{attribute 'GeneratedUsingTerminal: EL3064-0000-0020'}
{attribute addProperty BoxType "EL3064-0000-0020"}
{attribute addProperty Id "WcStateAT %I*BOOL1InputToggleAT %I*BOOL1"}
{attribute addProperty CRC "2425479403"}
{attribute addProperty Size "2"}
TYPE WcState_9091E0EB :
STRUCT
	{attribute addProperty Name "WcState"}
	WcState AT %I* : BOOL;
	{attribute addProperty Name "InputToggle"}
	InputToggle AT %I* : BOOL;
END_STRUCT
END_TYPE

(* stored: Version 1.2.0.0, ProductVersion 3.1.4024.9
   DUT WcState_9091E0EB: Id {ddc7b955-347c-4e5e-88fe-01aa397d0dd6} *)
